// SIMATIC S7-200 project (STEP 7-Micro/WIN), CPU 221 REL 01.10

ORGANIZATION_BLOCK 主程序:OB1
TITLE=程序注释
BEGIN
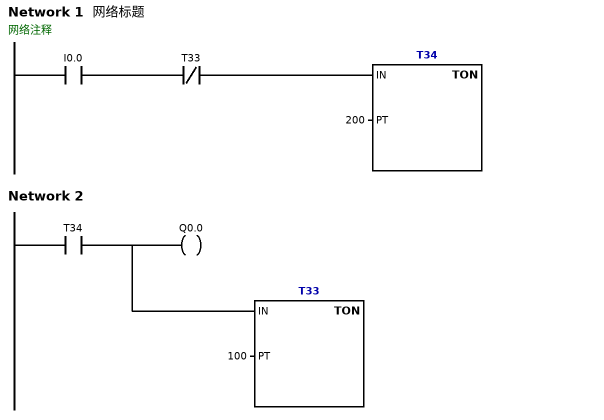
Network 1 // 网络标题
// 网络注释
LD     I0.0
AN     T33
TON    T34, 200
Network 2
LD     T34
=      Q0.0
TON    T33, 100
END_ORGANIZATION_BLOCK
